{attribute 'linkalways'} 
{attribute 'no_explicit_call' := 'This FB is a CLASS and must be accessed using methods or properties'}
{attribute 'enable_dynamic_creation'}
FUNCTION_BLOCK _ETcVnFlipAxis EXTENDS EnumDatatypeBase
VAR
	localData : ETcVnFlipAxis;
	activeData : REFERENCE TO ETcVnFlipAxis;
	enumBaseDatatype : _INT(localData);
END_VAR

METHOD PRIVATE AddLocalEnumeration
VAR_INPUT
	Enumeration : T_MAXSTRING;
	Value : ETcVnFlipAxis;
END_VAR
AddEnumeration(Enumeration, Value);
END_METHOD

PROPERTY PUBLIC Address : PVOID
GET
Address := ADR(activeData);
END_GET
END_PROPERTY

METHOD PUBLIC ClearReference
VAR_INPUT
END_VAR
activeData REF= localData;
SetBaseDatatypeReference();
END_METHOD

METHOD PUBLIC Clone : I_Datatype
VAR
    pClone : POINTER TO _ETcVnFlipAxis;
END_VAR
pClone := __NEW(_ETcVnFlipAxis(InitialValue := Value));
Clone := pClone^;
END_METHOD

METHOD FB_init : BOOL
VAR_INPUT
	bInitRetains : BOOL; // if TRUE, the retain variables are initialized (warm start / cold start)
	bInCopyCode : BOOL;  // if TRUE, the instance afterwards gets moved into the copy code (online change)
	InitialValue : ETcVnFlipAxis;
END_VAR
localData := InitialValue;
AddBaseDatatype(enumBaseDatatype);
ClearReference();

AddLocalEnumeration('TCVN_FA_XY', ETcVnFlipAxis.TCVN_FA_XY);
AddLocalEnumeration('TCVN_FA_X', ETcVnFlipAxis.TCVN_FA_X);
AddLocalEnumeration('TCVN_FA_Y', ETcVnFlipAxis.TCVN_FA_Y);
END_METHOD

PROPERTY PUBLIC Identifier : T_MAXSTRING
GET
Identifier := 'ETcVnFlipAxis';
END_GET
END_PROPERTY

METHOD IsEnumeratorValueEqual : BOOL
VAR_INPUT
	Enumerator : I_KeyValueForwardEnumerator;
END_VAR
VAR
	storedValue : ETcVnFlipAxis;
END_VAR
IF NOT Enumerator.TryGet(storedValue) THEN
	RETURN;
END_IF

IsEnumeratorValueEqual := storedValue = activeData;
END_METHOD

METHOD PUBLIC MakeReferenceTo
VAR_INPUT
	ReferenceTarget : REFERENCE TO ETcVnFlipAxis;
END_VAR
activeData REF= ReferenceTarget;
SetBaseDatatypeReference();
END_METHOD

METHOD PROTECTED SetBaseDatatypeReference
VAR_INPUT
END_VAR
enumBaseDatatype.MakeReferenceTo(activeData);
END_METHOD

PROPERTY PUBLIC Size : UDINT
GET
Size := SIZEOF(activeData);
END_GET
END_PROPERTY

METHOD TryMakeReferenceTo : BOOL
VAR_INPUT
	Target : I_Datatype;
END_VAR
VAR
	targetAsEnum : I_EnumDatatype;
	pTargetData : POINTER TO ETcVnFlipAxis;
END_VAR
IF NOT Target.TryResolveAsEnumDatatype(targetAsEnum) THEN
	RETURN;
END_IF

IF targetAsEnum.Identifier <> Identifier THEN
	RETURN;
END_IF

pTargetData := Target.Address;
activeData REF= pTargetData^;
SetBaseDatatypeReference();
TryMakeReferenceTo := TRUE;
END_METHOD

PROPERTY PUBLIC Value : ETcVnFlipAxis
GET
Value := activeData;
END_GET
SET
activeData := Value;
END_SET
END_PROPERTY

END_FUNCTION_BLOCK

(* stored: Version 1.1.0.1, ProductVersion 3.1.4024.12
   POU _ETcVnFlipAxis: Id {5c294a5b-bb24-4409-b86f-593716524bdc}, SpecialFunc None
   Folder Constructor: Id {24caa4d9-c587-4c73-96a2-9eacdb13d9e1}
   Folder Private: Id {8917fead-1c19-41f3-99bf-7e3eebbd1a7b}
   Folder Protected: Id {d22cd535-c0eb-494d-bfb4-aceaa7fcfa5b}
   Method AddLocalEnumeration: Id {132c18ac-bb95-4382-9086-b5fd9b5b6e56}
   Property Address: Id {3cce8095-8c68-4033-bbfb-4a2bd19ed432}
   Get Get: Id {058a4cdc-a36a-4610-9d11-5c5ba0f7c504}
   Method ClearReference: Id {55f5a47c-1b16-484b-b50b-2e4fc296e3b0}
   Method Clone: Id {ba19e4c3-fd9b-47c1-a2a0-b6d0f246b043}
   Method FB_init: Id {7ef3f3ef-046d-48a7-aa61-d1a9da2e7e2d}
   Property Identifier: Id {acb7e7b2-fdca-459f-aaa2-bbe54731a5a8}
   Get Get: Id {d518971c-dc39-4606-a397-dedd8d4dbbab}
   Method IsEnumeratorValueEqual: Id {6796c369-9398-45f6-b1d2-44c0716d85bd}
   Method MakeReferenceTo: Id {f4daf9c8-392a-490a-ad01-a8f495eb40f0}
   Method SetBaseDatatypeReference: Id {cc4a7a5e-8693-43b0-9fa9-5dcfd0ede578}
   Property Size: Id {dc1874ba-2dee-4354-ae2b-d548e86ef444}
   Get Get: Id {8417124a-1b27-46da-8b98-3fd6d510f2ac}
   Method TryMakeReferenceTo: Id {83e345fa-916e-4f5f-af2b-d9b3b0866026}
   Property Value: Id {66e77848-6b5a-4122-ae7b-e473dee30011}
   Get Get: Id {0ccaa258-67da-438f-87b2-b78197c4eea3}
   Set Set: Id {7405ee18-b6f5-43d9-9418-1198518622cd} *)
